(* Logix 5000 project; controller SX_V040001_C001 vendor 1 type 14 code 77 rev 16.22; software revision 16.04; part 22 of 35 *)
(* tags used below, declared in another part *)
   ALL_KINDS : INT[90];
   CMD : INT[36];
   command_number : INT;
   command_type : DINT;
   command_value : INT;
   DATAOP : INT[10];
   DRIVE : INT[32];
   G_DInput : DINT[3];
   G_DOutput : DINT[3];
   louvre : INT[11];
   m_alarm_exist : BOOL;
   METERING : INT[44];
   METERING_PULSE : DINT[14];
   NOTDOS : INT[6];
   PARAM_VISIWIN_PART_1 : INT[101];
   PARAM_VISIWIN_PART_2 : INT[100];
   PARAM_VISIWIN_PART_3 : INT[100];
   PARAM_VISIWIN_PART_4 : INT[100];
   PARAM_VISIWIN_PART_5 : INT[100];
   PARAMETER : INT[501];
   RECIPE_GENERAL : INT[405];
   RECIPE_VISIWIN_PART_1 : INT[100];
   RECIPE_VISIWIN_PART_2 : INT[100];
   RECIPE_VISIWIN_PART_3 : INT[100];
   RECIPE_VISIWIN_PART_4 : INT[100];
   RECIPE_VISIWIN_PART_5 : INT[5];
   RM_CMD : INT[9];
(* MainProgram, continued *)

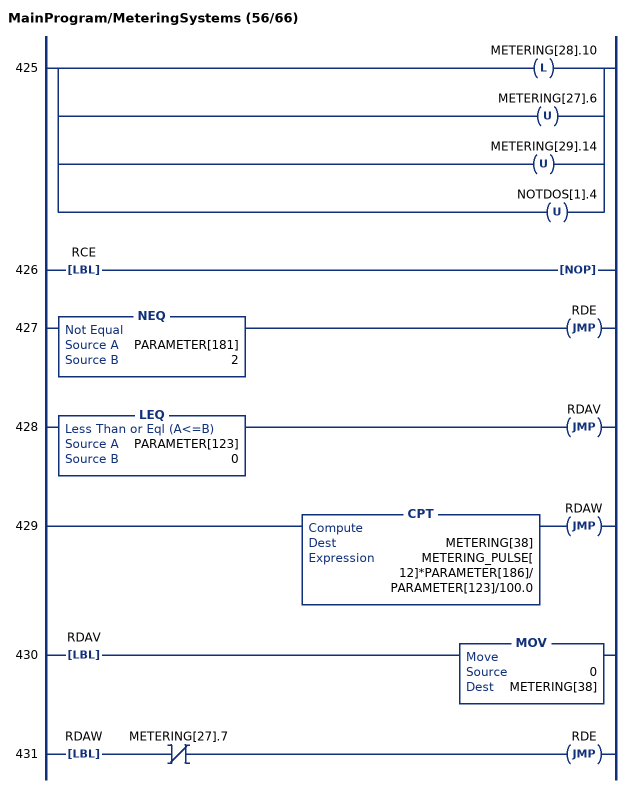
   [picture p477: MainProgram/MeteringSystems rungs 425-431]
   425: [OTL(METERING[28].10) ,OTU(METERING[27].6) ,OTU(METERING[29].14) ,OTU(NOTDOS[1].4) ];
   426: LBL(RCE)NOP();
   427: NEQ(PARAMETER[181],2)JMP(RDE);
   428: LEQ(PARAMETER[123],0)JMP(RDAV);
   429: CPT(METERING[38],METERING_PULSE[12]*PARAMETER[186]/PARAMETER[123]/100.0)JMP(RDAW);
   430: LBL(RDAV)MOV(0,METERING[38]);
   431: LBL(RDAW)XIO(METERING[27].7)JMP(RDE);
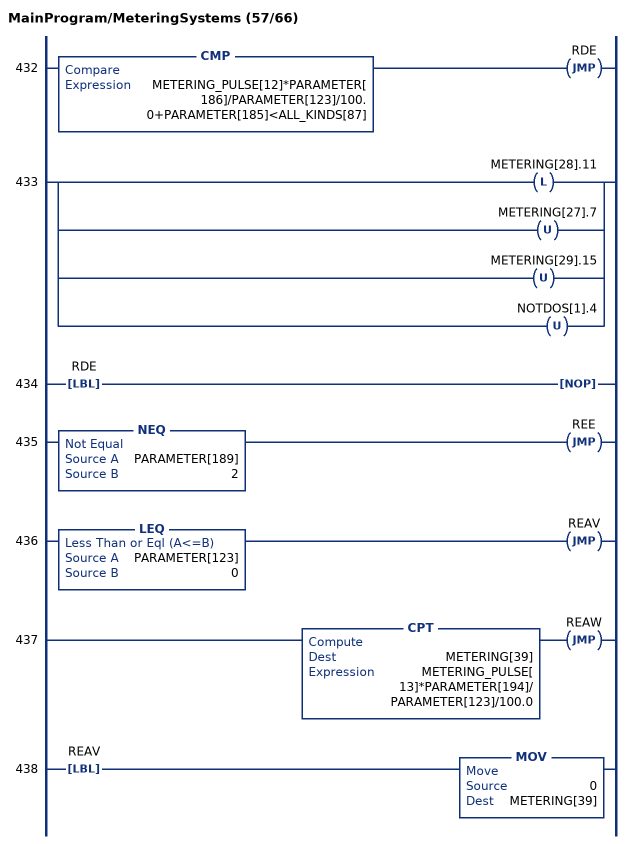
   432: CMP(METERING_PULSE[12]*PARAMETER[186]/PARAMETER[123]/100.0+PARAMETER[185]<ALL_KINDS[87])JMP(RDE);
   433: [OTL(METERING[28].11) ,OTU(METERING[27].7) ,OTU(METERING[29].15) ,OTU(NOTDOS[1].4) ];
   434: LBL(RDE)NOP();
   435: NEQ(PARAMETER[189],2)JMP(REE);
   436: LEQ(PARAMETER[123],0)JMP(REAV);
   437: CPT(METERING[39],METERING_PULSE[13]*PARAMETER[194]/PARAMETER[123]/100.0)JMP(REAW);
   438: LBL(REAV)MOV(0,METERING[39]);
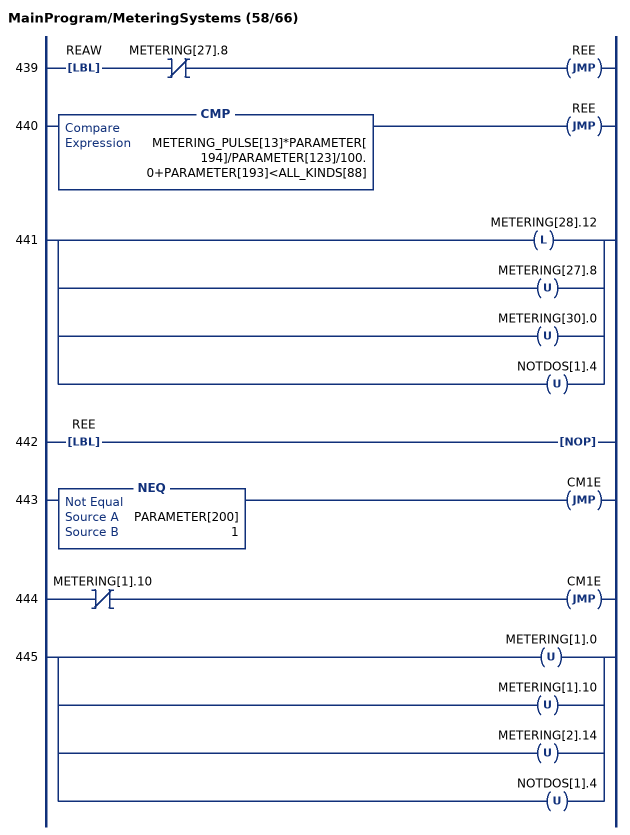
   439: LBL(REAW)XIO(METERING[27].8)JMP(REE);
   440: CMP(METERING_PULSE[13]*PARAMETER[194]/PARAMETER[123]/100.0+PARAMETER[193]<ALL_KINDS[88])JMP(REE);
   441: [OTL(METERING[28].12) ,OTU(METERING[27].8) ,OTU(METERING[30].0) ,OTU(NOTDOS[1].4) ];
   442: LBL(REE)NOP();
   443: NEQ(PARAMETER[200],1)JMP(CM1E);
   444: XIO(METERING[1].10)JMP(CM1E);
   445: [OTU(METERING[1].0) ,OTU(METERING[1].10) ,OTU(METERING[2].14) ,OTU(NOTDOS[1].4) ];
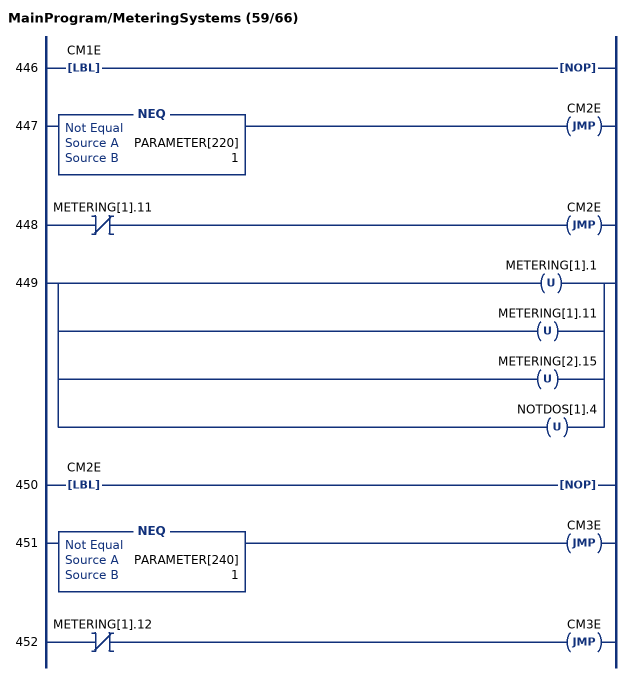
   446: LBL(CM1E)NOP();
   447: NEQ(PARAMETER[220],1)JMP(CM2E);
   448: XIO(METERING[1].11)JMP(CM2E);
   449: [OTU(METERING[1].1) ,OTU(METERING[1].11) ,OTU(METERING[2].15) ,OTU(NOTDOS[1].4) ];
   450: LBL(CM2E)NOP();
   451: NEQ(PARAMETER[240],1)JMP(CM3E);
   452: XIO(METERING[1].12)JMP(CM3E);
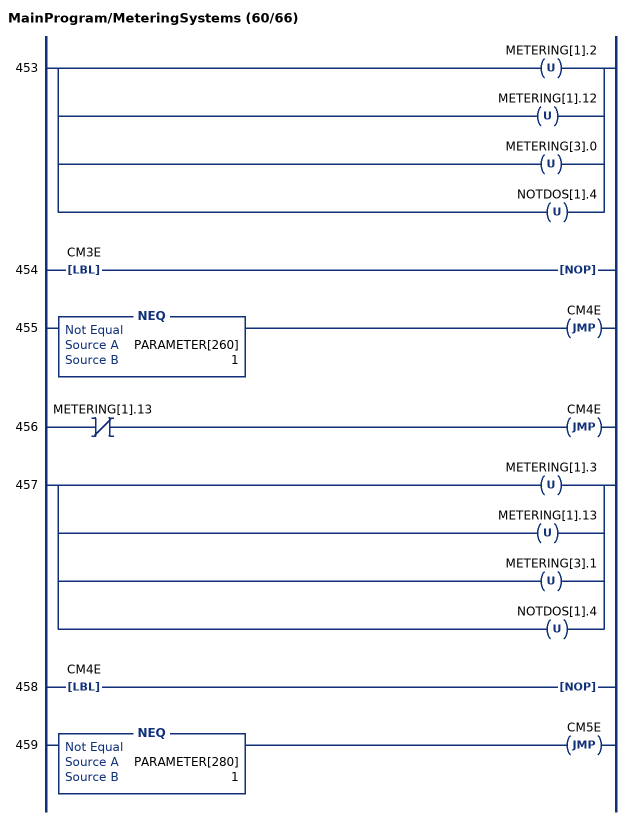
   453: [OTU(METERING[1].2) ,OTU(METERING[1].12) ,OTU(METERING[3].0) ,OTU(NOTDOS[1].4) ];
   454: LBL(CM3E)NOP();
   455: NEQ(PARAMETER[260],1)JMP(CM4E);
   456: XIO(METERING[1].13)JMP(CM4E);
   457: [OTU(METERING[1].3) ,OTU(METERING[1].13) ,OTU(METERING[3].1) ,OTU(NOTDOS[1].4) ];
   458: LBL(CM4E)NOP();
   459: NEQ(PARAMETER[280],1)JMP(CM5E);
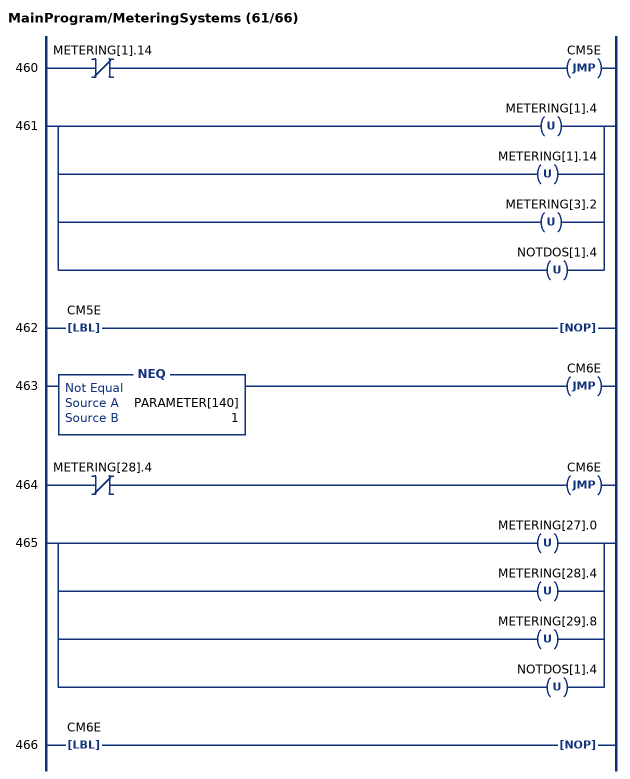
   460: XIO(METERING[1].14)JMP(CM5E);
   461: [OTU(METERING[1].4) ,OTU(METERING[1].14) ,OTU(METERING[3].2) ,OTU(NOTDOS[1].4) ];
   462: LBL(CM5E)NOP();
   463: NEQ(PARAMETER[140],1)JMP(CM6E);
   464: XIO(METERING[28].4)JMP(CM6E);
   465: [OTU(METERING[27].0) ,OTU(METERING[28].4) ,OTU(METERING[29].8) ,OTU(NOTDOS[1].4) ];
   466: LBL(CM6E)NOP();
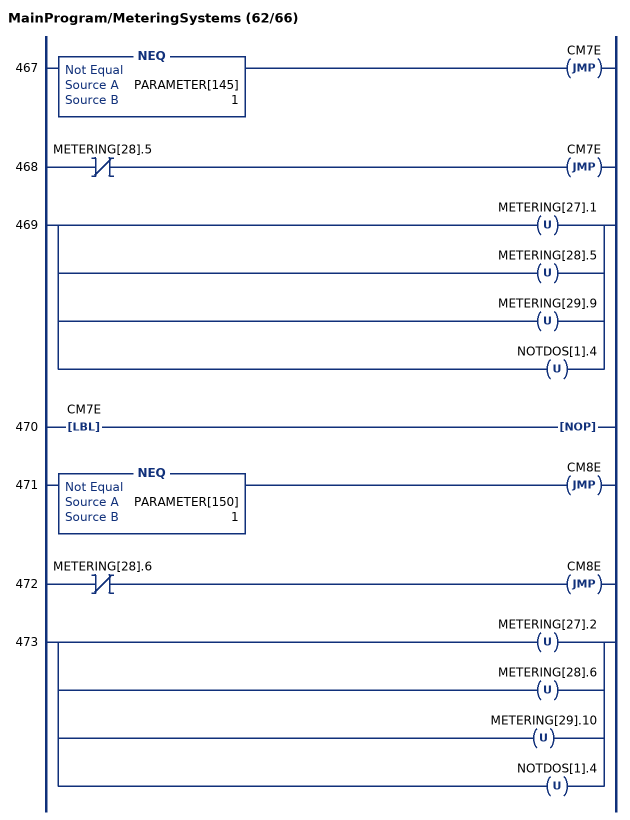
   467: NEQ(PARAMETER[145],1)JMP(CM7E);
   468: XIO(METERING[28].5)JMP(CM7E);
   469: [OTU(METERING[27].1) ,OTU(METERING[28].5) ,OTU(METERING[29].9) ,OTU(NOTDOS[1].4) ];
   470: LBL(CM7E)NOP();
   471: NEQ(PARAMETER[150],1)JMP(CM8E);
   472: XIO(METERING[28].6)JMP(CM8E);
   473: [OTU(METERING[27].2) ,OTU(METERING[28].6) ,OTU(METERING[29].10) ,OTU(NOTDOS[1].4) ];
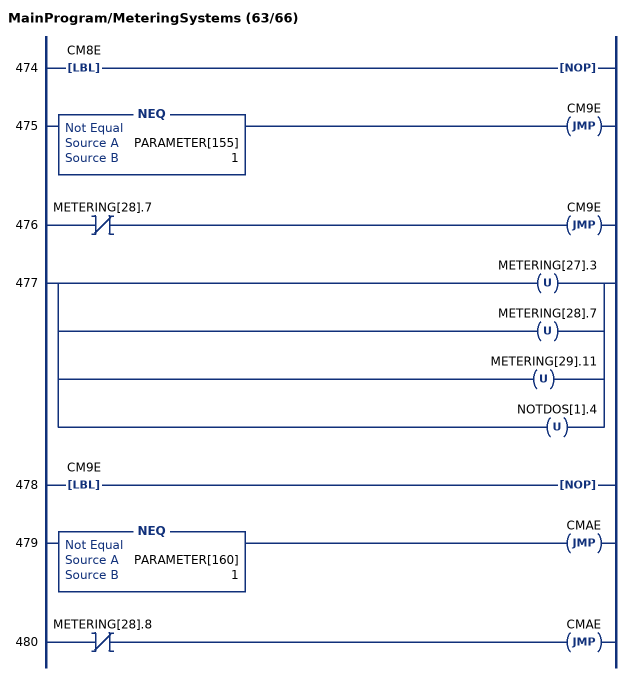
   474: LBL(CM8E)NOP();
   475: NEQ(PARAMETER[155],1)JMP(CM9E);
   476: XIO(METERING[28].7)JMP(CM9E);
   477: [OTU(METERING[27].3) ,OTU(METERING[28].7) ,OTU(METERING[29].11) ,OTU(NOTDOS[1].4) ];
   478: LBL(CM9E)NOP();
   479: NEQ(PARAMETER[160],1)JMP(CMAE);
   480: XIO(METERING[28].8)JMP(CMAE);
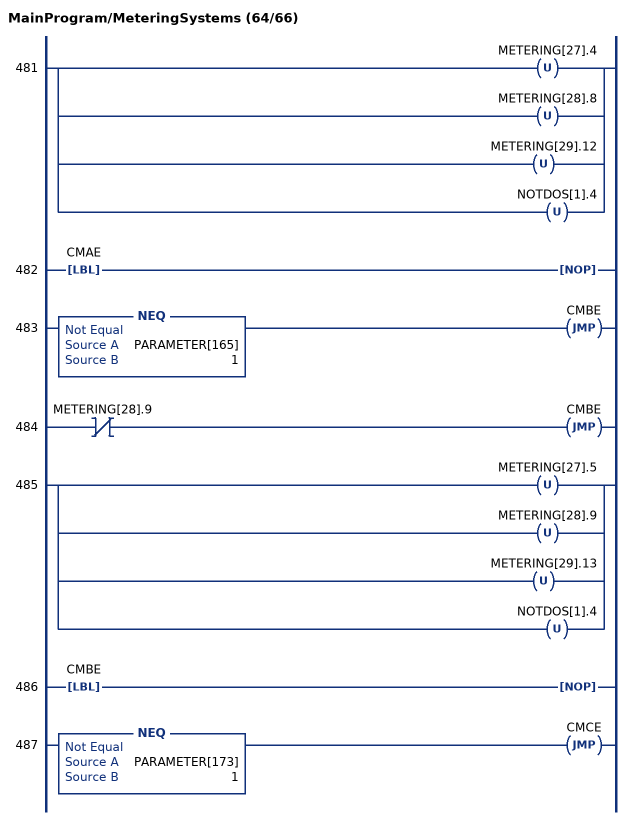
   481: [OTU(METERING[27].4) ,OTU(METERING[28].8) ,OTU(METERING[29].12) ,OTU(NOTDOS[1].4) ];
   482: LBL(CMAE)NOP();
   483: NEQ(PARAMETER[165],1)JMP(CMBE);
   484: XIO(METERING[28].9)JMP(CMBE);
   485: [OTU(METERING[27].5) ,OTU(METERING[28].9) ,OTU(METERING[29].13) ,OTU(NOTDOS[1].4) ];
   486: LBL(CMBE)NOP();
   487: NEQ(PARAMETER[173],1)JMP(CMCE);
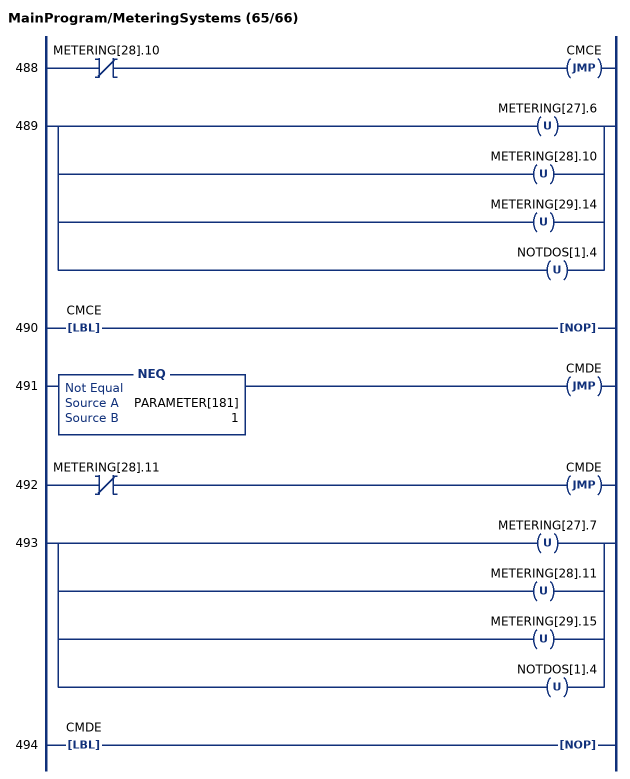
   488: XIO(METERING[28].10)JMP(CMCE);
   489: [OTU(METERING[27].6) ,OTU(METERING[28].10) ,OTU(METERING[29].14) ,OTU(NOTDOS[1].4) ];
   490: LBL(CMCE)NOP();
   491: NEQ(PARAMETER[181],1)JMP(CMDE);
   492: XIO(METERING[28].11)JMP(CMDE);
   493: [OTU(METERING[27].7) ,OTU(METERING[28].11) ,OTU(METERING[29].15) ,OTU(NOTDOS[1].4) ];
   494: LBL(CMDE)NOP();
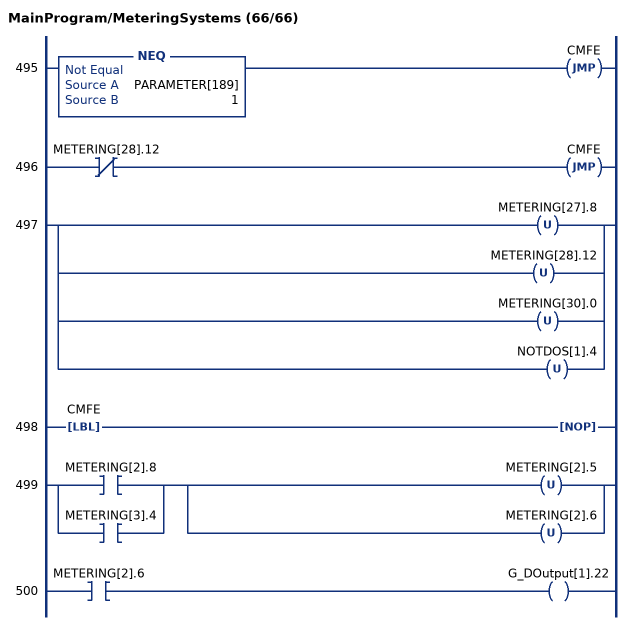
   495: NEQ(PARAMETER[189],1)JMP(CMFE);
   496: XIO(METERING[28].12)JMP(CMFE);
   497: [OTU(METERING[27].8) ,OTU(METERING[28].12) ,OTU(METERING[30].0) ,OTU(NOTDOS[1].4) ];
   498: LBL(CMFE)NOP();
   499: [XIC(METERING[2].8) ,XIC(METERING[3].4) ][OTU(METERING[2].5) ,OTU(METERING[2].6) ];
   500: XIC(METERING[2].6)OTE(G_DOutput[1].22);
END_ROUTINE

ROUTINE OP_Handler_VisiWin   (* ladder *)
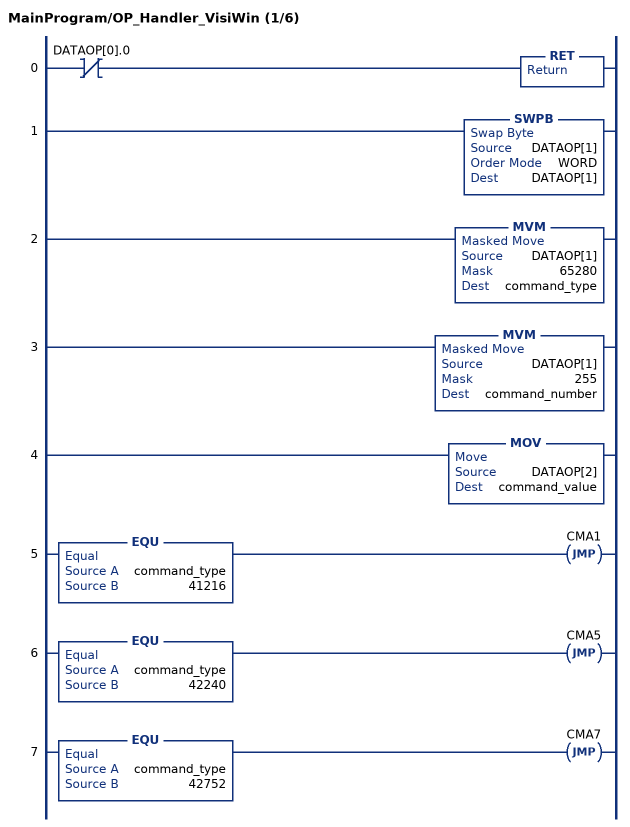
   0: XIO(DATAOP[0].0)RET();
   1: SWPB(DATAOP[1],WORD,DATAOP[1]);
   2: MVM(DATAOP[1],65280,command_type);
   3: MVM(DATAOP[1],255,command_number);
   4: MOV(DATAOP[2],command_value);
   5: EQU(command_type,41216)JMP(CMA1);
   6: EQU(command_type,42240)JMP(CMA5);
   7: EQU(command_type,42752)JMP(CMA7);
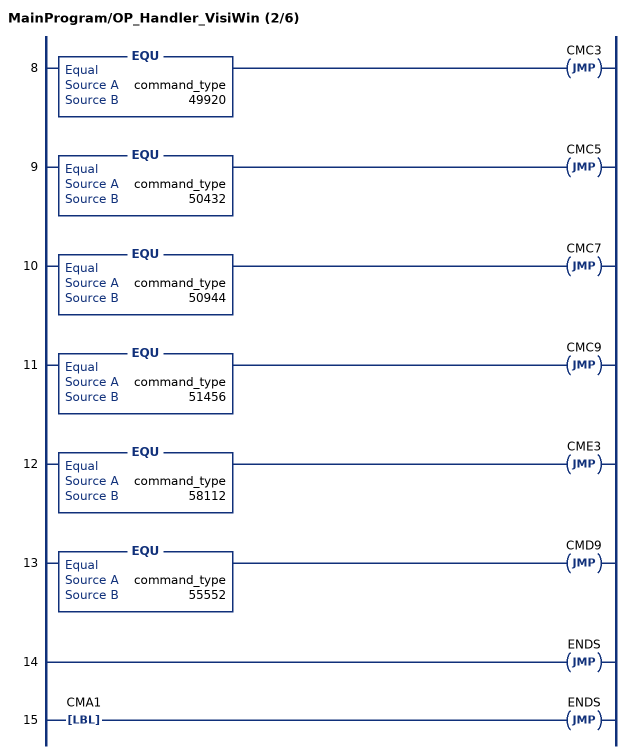
   8: EQU(command_type,49920)JMP(CMC3);
   9: EQU(command_type,50432)JMP(CMC5);
   10: EQU(command_type,50944)JMP(CMC7);
   11: EQU(command_type,51456)JMP(CMC9);
   12: EQU(command_type,58112)JMP(CME3);
   13: EQU(command_type,55552)JMP(CMD9);
   14: JMP(ENDS);
   15: LBL(CMA1)JMP(ENDS);
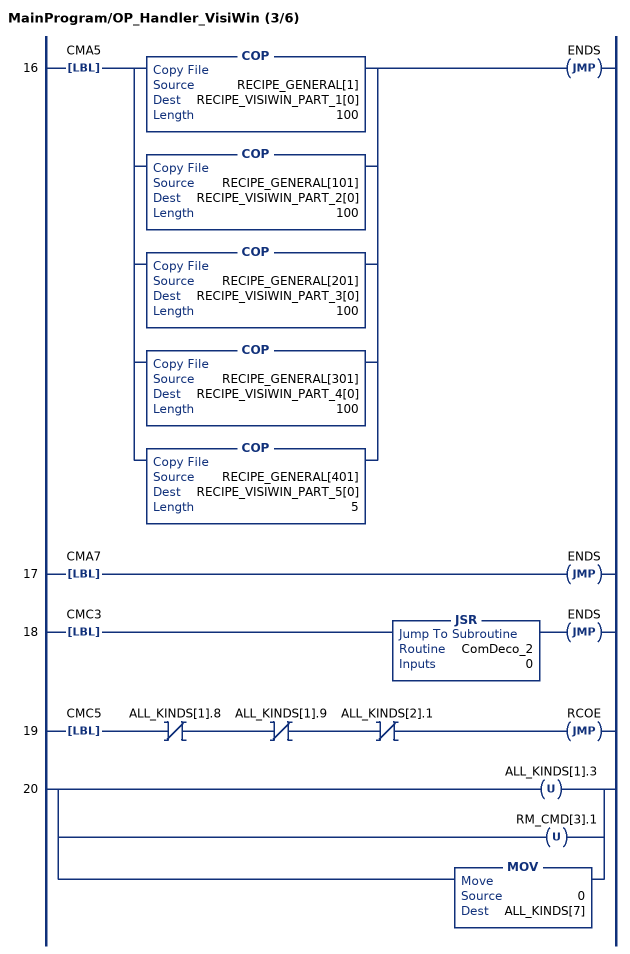
   16: LBL(CMA5)[COP(RECIPE_GENERAL[1],RECIPE_VISIWIN_PART_1[0],100) ,COP(RECIPE_GENERAL[101],RECIPE_VISIWIN_PART_2[0],100) ,COP(RECIPE_GENERAL[201],RECIPE_VISIWIN_PART_3[0],100) ,COP(RECIPE_GENERAL[301],RECIPE_VISIWIN_PART_4[0],100) ,COP(RECIPE_GENERAL[401],RECIPE_VISIWIN_PART_5[0],5) ]JMP(ENDS);
   17: LBL(CMA7)JMP(ENDS);
   18: LBL(CMC3)JSR(ComDeco_2,0)JMP(ENDS);
   19: LBL(CMC5)XIO(ALL_KINDS[1].8)XIO(ALL_KINDS[1].9)XIO(ALL_KINDS[2].1)JMP(RCOE);
   20: [OTU(ALL_KINDS[1].3) ,OTU(RM_CMD[3].1) ,MOV(0,ALL_KINDS[7]) ];
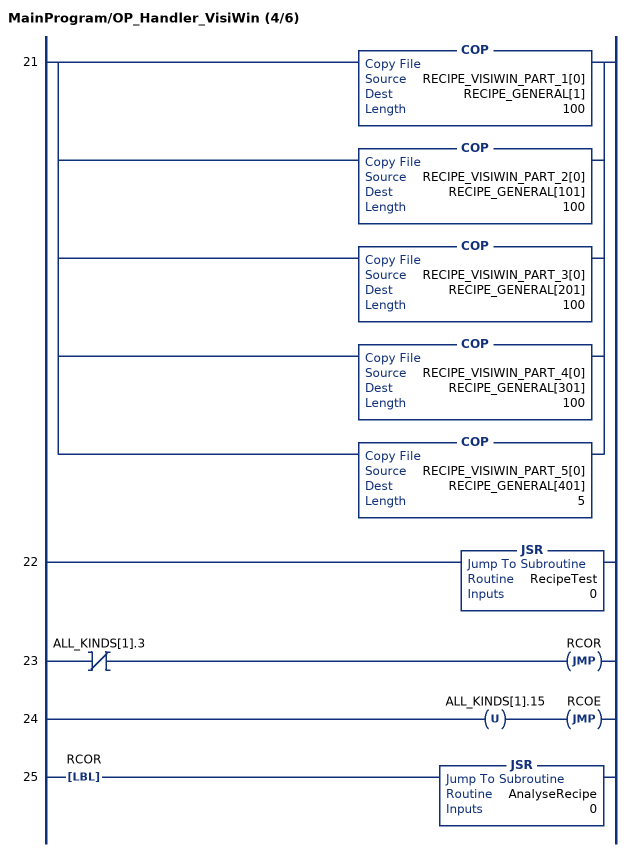
   21: [COP(RECIPE_VISIWIN_PART_1[0],RECIPE_GENERAL[1],100) ,COP(RECIPE_VISIWIN_PART_2[0],RECIPE_GENERAL[101],100) ,COP(RECIPE_VISIWIN_PART_3[0],RECIPE_GENERAL[201],100) ,COP(RECIPE_VISIWIN_PART_4[0],RECIPE_GENERAL[301],100) ,COP(RECIPE_VISIWIN_PART_5[0],RECIPE_GENERAL[401],5) ];
   22: JSR(RecipeTest,0);
   23: XIO(ALL_KINDS[1].3)JMP(RCOR);
   24: OTU(ALL_KINDS[1].15)JMP(RCOE);
   25: LBL(RCOR)JSR(AnalyseRecipe,0);
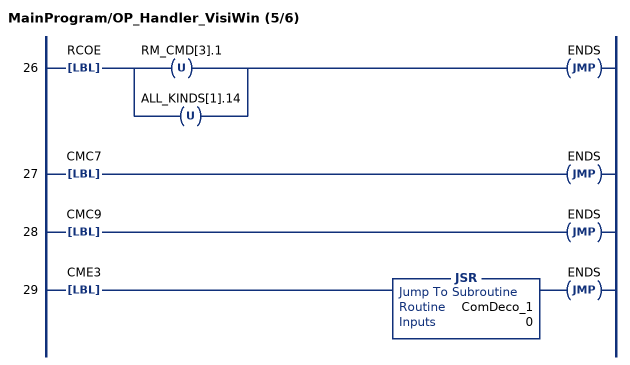
   26: LBL(RCOE)[OTU(RM_CMD[3].1) ,OTU(ALL_KINDS[1].14) ]JMP(ENDS);
   27: LBL(CMC7)JMP(ENDS);
   28: LBL(CMC9)JMP(ENDS);
   29: LBL(CME3)JSR(ComDeco_1,0)JMP(ENDS);
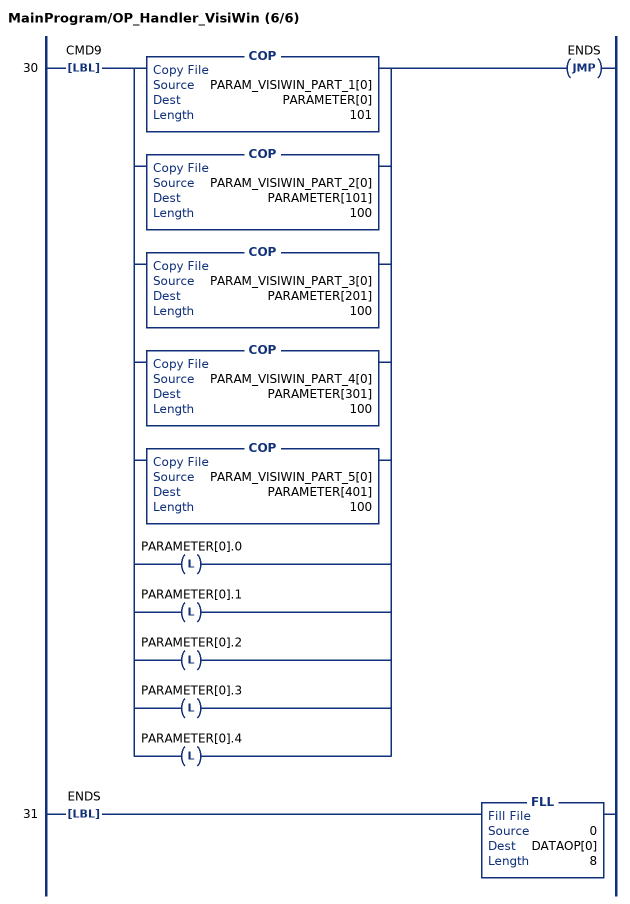
   30: LBL(CMD9)[COP(PARAM_VISIWIN_PART_1[0],PARAMETER[0],101) ,COP(PARAM_VISIWIN_PART_2[0],PARAMETER[101],100) ,COP(PARAM_VISIWIN_PART_3[0],PARAMETER[201],100) ,COP(PARAM_VISIWIN_PART_4[0],PARAMETER[301],100) ,COP(PARAM_VISIWIN_PART_5[0],PARAMETER[401],100) ,OTL(PARAMETER[0].0) ,OTL(PARAMETER[0].1) ,OTL(PARAMETER[0].2) ,OTL(PARAMETER[0].3) ,OTL(PARAMETER[0].4) ]JMP(ENDS);
   31: LBL(ENDS)FLL(0,DATAOP[0],8);
END_ROUTINE

ROUTINE OPC_Commands   (* ladder *)
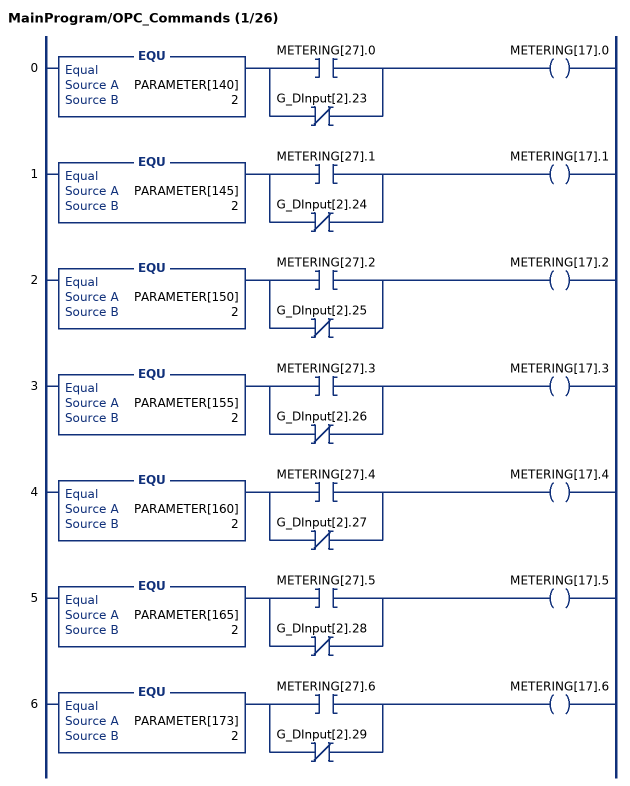
   0: EQU(PARAMETER[140],2)[XIC(METERING[27].0) ,XIO(G_DInput[2].23) ]OTE(METERING[17].0);
   1: EQU(PARAMETER[145],2)[XIC(METERING[27].1) ,XIO(G_DInput[2].24) ]OTE(METERING[17].1);
   2: EQU(PARAMETER[150],2)[XIC(METERING[27].2) ,XIO(G_DInput[2].25) ]OTE(METERING[17].2);
   3: EQU(PARAMETER[155],2)[XIC(METERING[27].3) ,XIO(G_DInput[2].26) ]OTE(METERING[17].3);
   4: EQU(PARAMETER[160],2)[XIC(METERING[27].4) ,XIO(G_DInput[2].27) ]OTE(METERING[17].4);
   5: EQU(PARAMETER[165],2)[XIC(METERING[27].5) ,XIO(G_DInput[2].28) ]OTE(METERING[17].5);
   6: EQU(PARAMETER[173],2)[XIC(METERING[27].6) ,XIO(G_DInput[2].29) ]OTE(METERING[17].6);
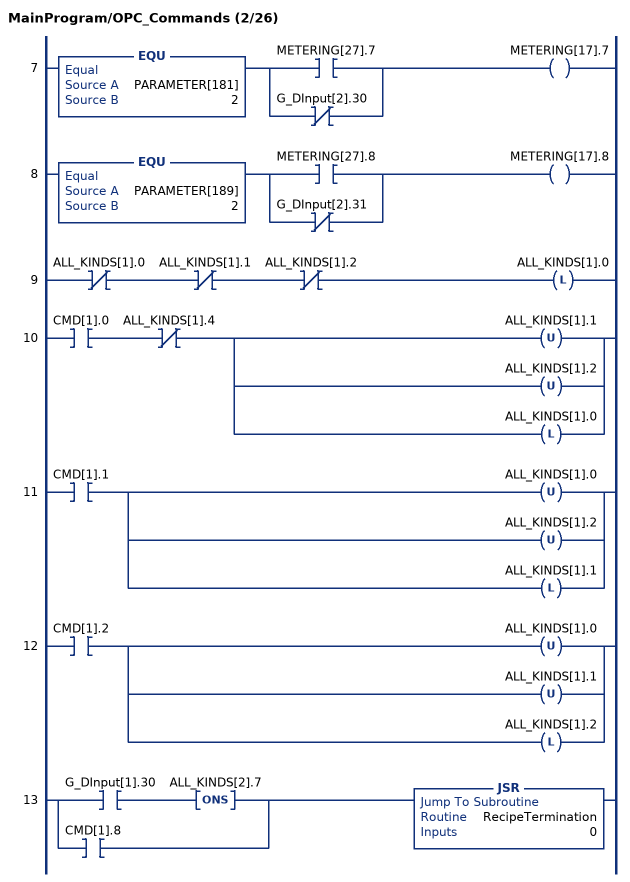
   7: EQU(PARAMETER[181],2)[XIC(METERING[27].7) ,XIO(G_DInput[2].30) ]OTE(METERING[17].7);
   8: EQU(PARAMETER[189],2)[XIC(METERING[27].8) ,XIO(G_DInput[2].31) ]OTE(METERING[17].8);
   9: XIO(ALL_KINDS[1].0)XIO(ALL_KINDS[1].1)XIO(ALL_KINDS[1].2)OTL(ALL_KINDS[1].0);
   10: XIC(CMD[1].0)XIO(ALL_KINDS[1].4)[OTU(ALL_KINDS[1].1) ,OTU(ALL_KINDS[1].2) ,OTL(ALL_KINDS[1].0) ];
   11: XIC(CMD[1].1)[OTU(ALL_KINDS[1].0) ,OTU(ALL_KINDS[1].2) ,OTL(ALL_KINDS[1].1) ];
   12: XIC(CMD[1].2)[OTU(ALL_KINDS[1].0) ,OTU(ALL_KINDS[1].1) ,OTL(ALL_KINDS[1].2) ];
   13: [XIC(G_DInput[1].30) ONS(ALL_KINDS[2].7) ,XIC(CMD[1].8) ]JSR(RecipeTermination,0);
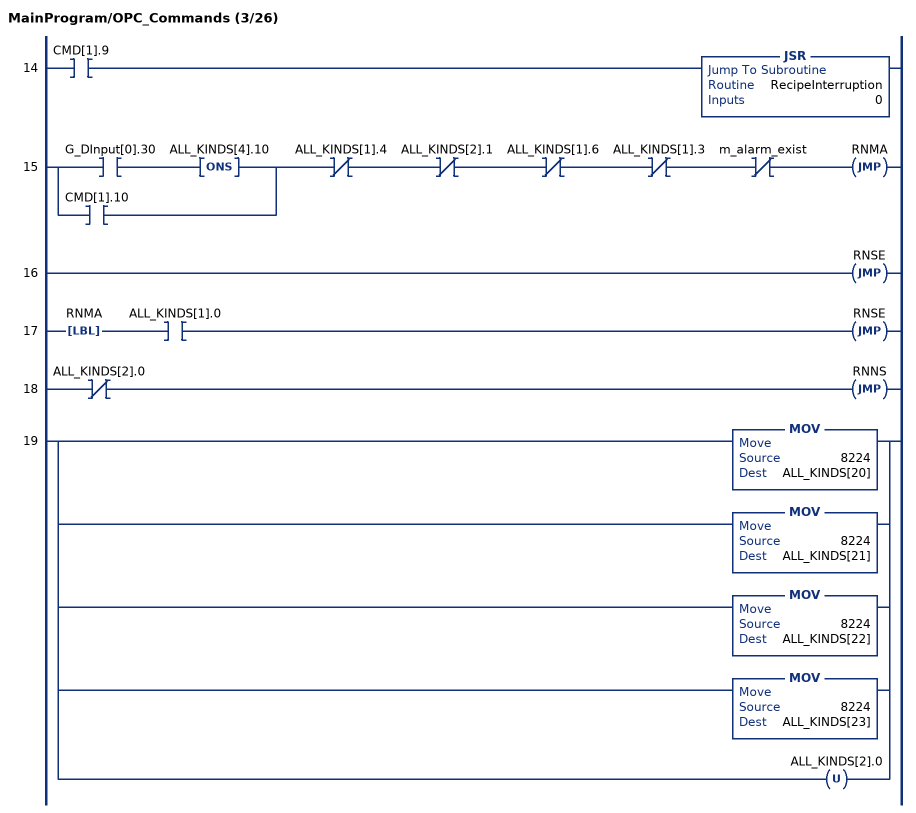
   14: XIC(CMD[1].9)JSR(RecipeInterruption,0);
   15: [XIC(G_DInput[0].30) ONS(ALL_KINDS[4].10) ,XIC(CMD[1].10) ]XIO(ALL_KINDS[1].4)XIO(ALL_KINDS[2].1)XIO(ALL_KINDS[1].6)XIO(ALL_KINDS[1].3)XIO(m_alarm_exist)JMP(RNMA);
   16: JMP(RNSE);
   17: LBL(RNMA)XIC(ALL_KINDS[1].0)JMP(RNSE);
   18: XIO(ALL_KINDS[2].0)JMP(RNNS);
   19: [MOV(8224,ALL_KINDS[20]) ,MOV(8224,ALL_KINDS[21]) ,MOV(8224,ALL_KINDS[22]) ,MOV(8224,ALL_KINDS[23]) ,OTU(ALL_KINDS[2].0) ];
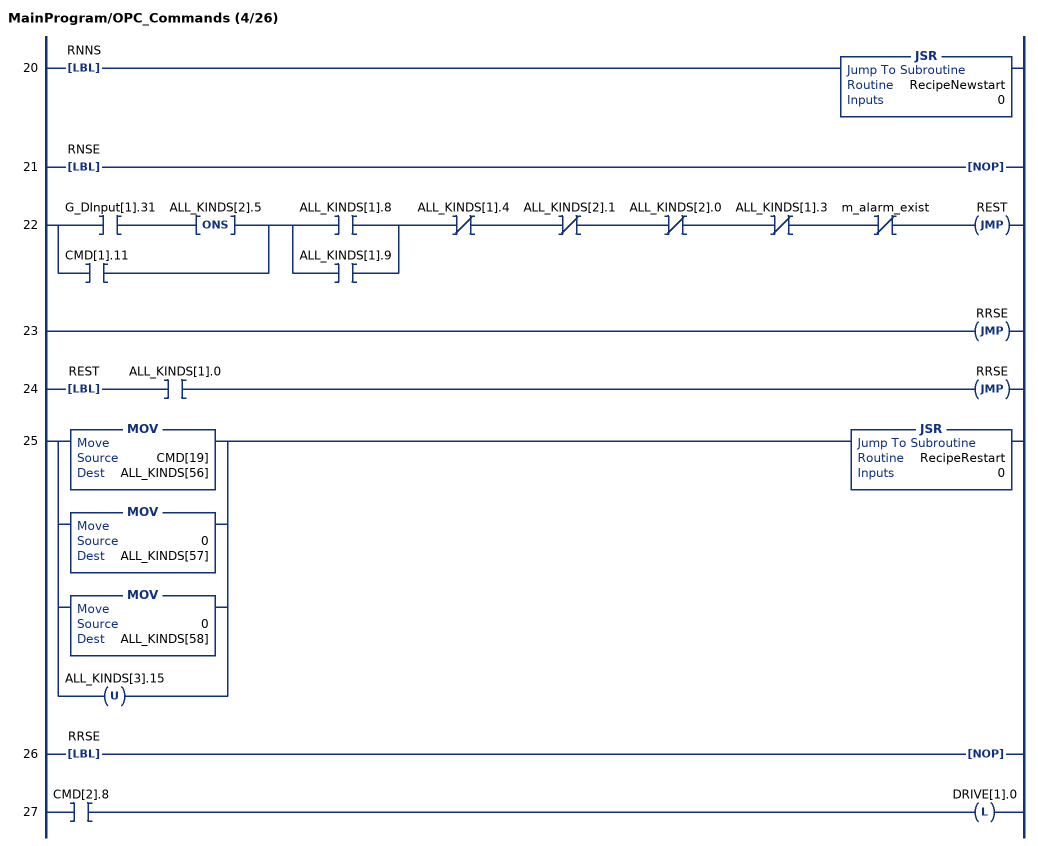
   20: LBL(RNNS)JSR(RecipeNewstart,0);
   21: LBL(RNSE)NOP();
   22: [XIC(G_DInput[1].31) ONS(ALL_KINDS[2].5) ,XIC(CMD[1].11) ][XIC(ALL_KINDS[1].8) ,XIC(ALL_KINDS[1].9) ]XIO(ALL_KINDS[1].4)XIO(ALL_KINDS[2].1)XIO(ALL_KINDS[2].0)XIO(ALL_KINDS[1].3)XIO(m_alarm_exist)JMP(REST);
   23: JMP(RRSE);
   24: LBL(REST)XIC(ALL_KINDS[1].0)JMP(RRSE);
   25: [MOV(CMD[19],ALL_KINDS[56]) ,MOV(0,ALL_KINDS[57]) ,MOV(0,ALL_KINDS[58]) ,OTU(ALL_KINDS[3].15) ]JSR(RecipeRestart,0);
   26: LBL(RRSE)NOP();
   27: XIC(CMD[2].8)OTL(DRIVE[1].0);
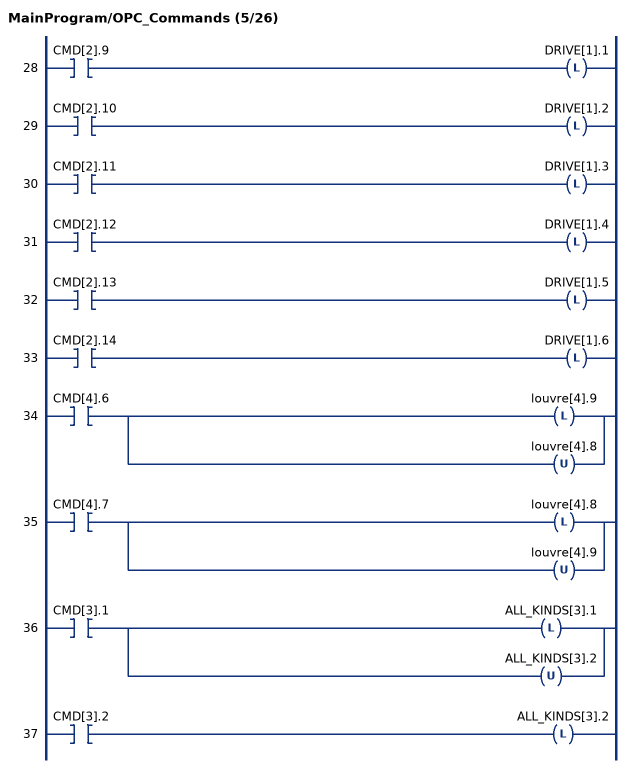
   28: XIC(CMD[2].9)OTL(DRIVE[1].1);
   29: XIC(CMD[2].10)OTL(DRIVE[1].2);
   30: XIC(CMD[2].11)OTL(DRIVE[1].3);
   31: XIC(CMD[2].12)OTL(DRIVE[1].4);
   32: XIC(CMD[2].13)OTL(DRIVE[1].5);
   33: XIC(CMD[2].14)OTL(DRIVE[1].6);
   34: XIC(CMD[4].6)[OTL(louvre[4].9) ,OTU(louvre[4].8) ];
   35: XIC(CMD[4].7)[OTL(louvre[4].8) ,OTU(louvre[4].9) ];
   36: XIC(CMD[3].1)[OTL(ALL_KINDS[3].1) ,OTU(ALL_KINDS[3].2) ];
   37: XIC(CMD[3].2)OTL(ALL_KINDS[3].2);
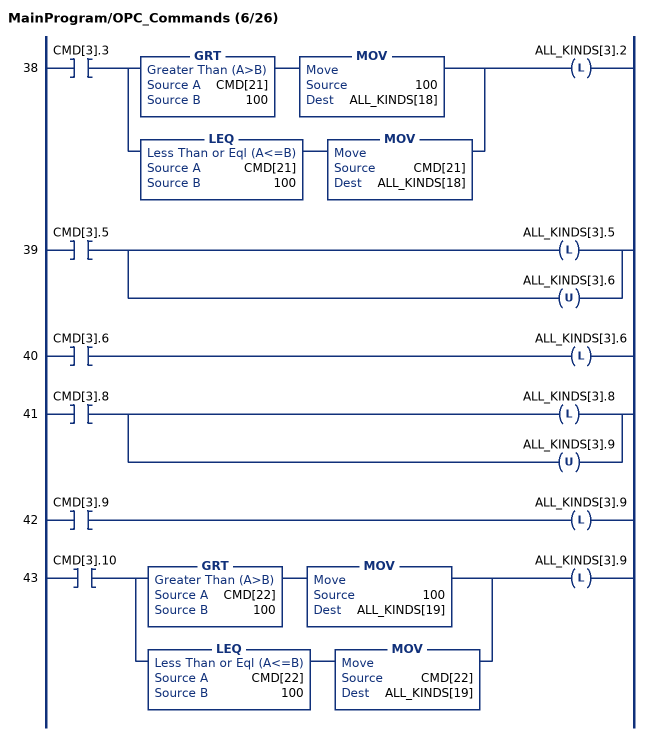
   38: XIC(CMD[3].3)[GRT(CMD[21],100) MOV(100,ALL_KINDS[18]) ,LEQ(CMD[21],100) MOV(CMD[21],ALL_KINDS[18]) ]OTL(ALL_KINDS[3].2);
   39: XIC(CMD[3].5)[OTL(ALL_KINDS[3].5) ,OTU(ALL_KINDS[3].6) ];
   40: XIC(CMD[3].6)OTL(ALL_KINDS[3].6);
   41: XIC(CMD[3].8)[OTL(ALL_KINDS[3].8) ,OTU(ALL_KINDS[3].9) ];
   42: XIC(CMD[3].9)OTL(ALL_KINDS[3].9);
   43: XIC(CMD[3].10)[GRT(CMD[22],100) MOV(100,ALL_KINDS[19]) ,LEQ(CMD[22],100) MOV(CMD[22],ALL_KINDS[19]) ]OTL(ALL_KINDS[3].9);
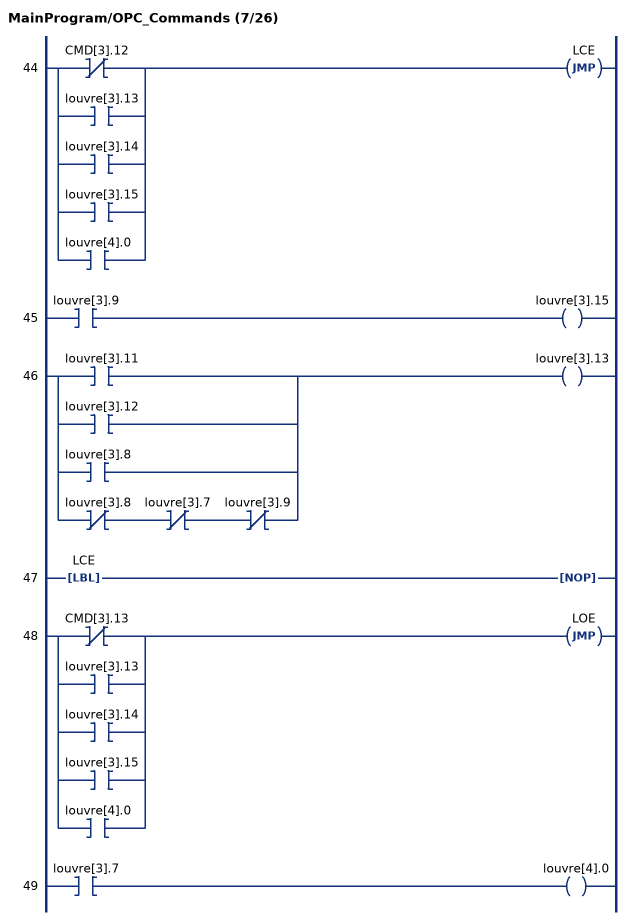
   44: [XIO(CMD[3].12) ,XIC(louvre[3].13) ,XIC(louvre[3].14) ,XIC(louvre[3].15) ,XIC(louvre[4].0) ]JMP(LCE);
   45: XIC(louvre[3].9)OTE(louvre[3].15);
   46: [XIC(louvre[3].11) ,XIC(louvre[3].12) ,XIC(louvre[3].8) ,XIO(louvre[3].8) XIO(louvre[3].7) XIO(louvre[3].9) ]OTE(louvre[3].13);
   47: LBL(LCE)NOP();
   48: [XIO(CMD[3].13) ,XIC(louvre[3].13) ,XIC(louvre[3].14) ,XIC(louvre[3].15) ,XIC(louvre[4].0) ]JMP(LOE);
   49: XIC(louvre[3].7)OTE(louvre[4].0);
